LIN {X 0,Y 107.094,Z 527.487,A -85,B 0,C 180,E1 -28422.092,E2 -28422.092} C_VEL
LIN {X 0,Y 108.586,Z 526.305,A -85,B 0,C 180,E1 -28423.07,E2 -28423.07} C_VEL
LIN {X 0,Y 109.785,Z 524.448,A -85,B 0,C 180,E1 -28426.243,E2 -28426.243} C_VEL
LIN {X 0,Y 110.569,Z 522.982,A -85,B 0,C 180,E1 -28429.008,E2 -28429.008} C_VEL
LIN {X 0,Y 111.254,Z 521.399,A -85,B 0,C 180,E1 -28432.742,E2 -28432.742} C_VEL
LIN {X 0,Y 111.93,Z 520.04,A -85,B 0,C 180,E1 -28436.401,E2 -28436.401} C_VEL
LIN {X 0,Y 112.516,Z 519.038,A -85,B 0,C 180,E1 -28440.001,E2 -28440.001} C_VEL
LIN {X 0,Y 112.419,Z 518.805,A -85,B 0,C 180,E1 -28443.585,E2 -28443.585} C_VEL
LIN {X 0,Y 112.118,Z 519.081,A -85,B 0,C 180,E1 -28447.203,E2 -28447.203} C_VEL
LIN {X 0,Y 111.817,Z 519.73,A -85,B 0,C 180,E1 -28450.869,E2 -28450.869} C_VEL
LIN {X 0,Y 111.466,Z 520.726,A -85,B 0,C 180,E1 -28454.609,E2 -28454.609} C_VEL
LIN {X 0,Y 110.518,Z 523.179,A -85,B 0,C 180,E1 -28460.473,E2 -28460.473} C_VEL
LIN {X 0,Y 109.085,Z 526.099,A -85,B 0,C 180,E1 -28465.582,E2 -28465.582} C_VEL
LIN {X 0,Y 107.757,Z 528.427,A -85,B 0,C 180,E1 -28469.143,E2 -28469.143} C_VEL
LIN {X 0,Y 106.14,Z 529.943,A -85,B 0,C 180,E1 -28470.596,E2 -28470.596} C_VEL
LIN {X 0,Y 100.627,Z 533.463,A -85,B 0,C 180,E1 -28473.059,E2 -28473.059} C_VEL
LIN {X 0,Y 92.597,Z 537.838,A -85,B 0,C 180,E1 -28477.165,E2 -28477.165} C_VEL
LIN {X 0,Y 85.11,Z 541.174,A -85,B 0,C 180,E1 -28481.997,E2 -28481.997} C_VEL
LIN {X 0,Y 76.203,Z 544.136,A -85,B 0,C 180,E1 -28489.79,E2 -28489.79} C_VEL
LIN {X 0,Y 72.407,Z 545.04,A -85,B 0,C 180,E1 -28494.382,E2 -28494.382} C_VEL
LIN {X 0,Y 69.095,Z 545.527,A -85,B 0,C 180,E1 -28499.43,E2 -28499.43} C_VEL
LIN {X 0,Y 64.573,Z 545.362,A -85,B 0,C 180,E1 -28510.942,E2 -28510.942} C_VEL
LIN {X 0,Y 62.726,Z 543.678,A -85,B 0,C 180,E1 -28523.566,E2 -28523.566} C_VEL
LIN {X 0,Y 62.673,Z 542.19,A -85,B 0,C 180,E1 -28529.999,E2 -28529.999} C_VEL
LIN {X 0,Y 62.878,Z 539.11,A -85,B 0,C 180,E1 -28539.65,E2 -28539.65} C_VEL
LIN {X 0,Y 64.442,Z 534.938,A -85,B 0,C 180,E1 -28549.096,E2 -28549.096} C_VEL
LIN {X 0,Y 68.08,Z 528.537,A -85,B 0,C 180,E1 -28559.361,E2 -28559.361} C_VEL
LIN {X 0,Y 72.709,Z 521.546,A -85,B 0,C 180,E1 -28567.164,E2 -28567.164} C_VEL
LIN {X 0,Y 76.458,Z 515.745,A -85,B 0,C 180,E1 -28571.951,E2 -28571.951} C_VEL
LIN {X 0,Y 80.603,Z 509.367,A -85,B 0,C 180,E1 -28575.998,E2 -28575.998} C_VEL
LIN {X 0,Y 82.695,Z 504.549,A -85,B 0,C 180,E1 -28578.958,E2 -28578.958} C_VEL
LIN {X 0,Y 85.692,Z 495.407,A -85,B 0,C 180,E1 -28584.098,E2 -28584.098} C_VEL
LIN {X 0,Y 87.474,Z 488.295,A -85,B 0,C 180,E1 -28587.735,E2 -28587.735} C_VEL
LIN {X 0,Y 86.8,Z 482.082,A -85,B 0,C 180,E1 -28592.382,E2 -28592.382} C_VEL
LIN {X 0,Y 85.779,Z 478.507,A -85,B 0,C 180,E1 -28595.816,E2 -28595.816} C_VEL
LIN {X 0,Y 84.988,Z 476.341,A -85,B 0,C 180,E1 -28598.152,E2 -28598.152} C_VEL
LIN {X 0,Y 83.456,Z 472.714,A -85,B 0,C 180,E1 -28602.857,E2 -28602.857} C_VEL
LIN {X 0,Y 81.455,Z 468.495,A -85,B 0,C 180,E1 -28610.062,E2 -28610.062} C_VEL
LIN {X 0,Y 80.014,Z 464.504,A -85,B 0,C 180,E1 -28619.999,E2 -28619.999} C_VEL
LIN {X 0,Y 79.435,Z 464.413,A -85,B 0,C 180,E1 -28630.191,E2 -28630.191} C_VEL
LIN {X 0,Y 79.756,Z 464.688,A -85,B 0,C 180,E1 -28634.24,E2 -28634.24} C_VEL
LIN {X 0,Y 80.144,Z 467.283,A -85,B 0,C 180,E1 -28640.534,E2 -28640.534} C_VEL
LIN {X 0,Y 81.313,Z 468.944,A -85,B 0,C 180,E1 -28645.604,E2 -28645.604} C_VEL
LIN {X 0,Y 83.366,Z 473.368,A -85,B 0,C 180,E1 -28653.224,E2 -28653.224} C_VEL
LIN {X 0,Y 85.065,Z 477.902,A -85,B 0,C 180,E1 -28658.853,E2 -28658.853} C_VEL
LIN {X 0,Y 86.341,Z 481.692,A -85,B 0,C 180,E1 -28662.899,E2 -28662.899} C_VEL
LIN {X 0,Y 87.659,Z 487.537,A -85,B 0,C 180,E1 -28668.17,E2 -28668.17} C_VEL
LIN {X 0,Y 87.904,Z 488.872,A -85,B 0,C 180,E1 -28669.284,E2 -28669.284} C_VEL
LIN {X 0,Y 86.406,Z 496.526,A -85,B 0,C 180,E1 -28673.867,E2 -28673.867} C_VEL
LIN {X 0,Y 86.132,Z 497.527,A -85,B 0,C 180,E1 -28674.455,E2 -28674.455} C_VEL
LIN {X 0,Y 81.043,Z 506.139,A -85,B 0,C 180,E1 -28678.648,E2 -28678.648} C_VEL
LIN {X 0,Y 75.891,Z 514.081,A -85,B 0,C 180,E1 -28683.905,E2 -28683.905} C_VEL
LIN {X 0,Y 70.618,Z 521.83,A -85,B 0,C 180,E1 -28691.13,E2 -28691.13} C_VEL
LIN {X 0,Y 67.264,Z 527.117,A -85,B 0,C 180,E1 -28697.94,E2 -28697.94} C_VEL
LIN {X 0,Y 64.323,Z 532.25,A -85,B 0,C 180,E1 -28706.87,E2 -28706.87} C_VEL
LIN {X 0,Y 63.116,Z 534.758,A -85,B 0,C 180,E1 -28712.542,E2 -28712.542} C_VEL
LIN {X 0,Y 61.74,Z 536.654,A -85,B 0,C 180,E1 -28717.534,E2 -28717.534} C_VEL
LIN {X 0,Y 58.637,Z 539.17,A -85,B 0,C 180,E1 -28726.171,E2 -28726.171} C_VEL
LIN {X 0,Y 56.92,Z 540.71,A -85,B 0,C 180,E1 -28733.757,E2 -28733.757} C_VEL
LIN {X 0,Y 56.998,Z 541.541,A -85,B 0,C 180,E1 -28739.685,E2 -28739.685} C_VEL
LIN {X 0,Y 57.396,Z 541.749,A -85,B 0,C 180,E1 -28741.62,E2 -28741.62} C_VEL
LIN {X 0,Y 61.763,Z 542.578,A -85,B 0,C 180,E1 -28753.058,E2 -28753.058} C_VEL
LIN {X 0,Y 66.596,Z 542.319,A -85,B 0,C 180,E1 -28760.716,E2 -28760.716} C_VEL
LIN {X 0,Y 73.961,Z 540.949,A -85,B 0,C 180,E1 -28768.783,E2 -28768.783} C_VEL
LIN {X 0,Y 81.011,Z 538.875,A -85,B 0,C 180,E1 -28774.294,E2 -28774.294} C_VEL
LIN {X 0,Y 89.976,Z 535.338,A -85,B 0,C 180,E1 -28779.605,E2 -28779.605} C_VEL
LIN {X 0,Y 99.681,Z 530.427,A -85,B 0,C 180,E1 -28783.96,E2 -28783.96} C_VEL
LIN {X 0,Y 101.944,Z 529.082,A -85,B 0,C 180,E1 -28784.828,E2 -28784.828} C_VEL
LIN {X 0,Y 103.445,Z 527.812,A -85,B 0,C 180,E1 -28786.652,E2 -28786.652} C_VEL
LIN {X 0,Y 105.01,Z 525.439,A -85,B 0,C 180,E1 -28792.308,E2 -28792.308} C_VEL
LIN {X 0,Y 105.847,Z 524.124,A -85,B 0,C 180,E1 -28796.194,E2 -28796.194} C_VEL
LIN {X 0,Y 106.629,Z 523.121,A -85,B 0,C 180,E1 -28800.001,E2 -28800.001} C_VEL
LIN {X 0,Y 106.581,Z 522.939,A -85,B 0,C 180,E1 -28803.782,E2 -28803.782} C_VEL
LIN {X 0,Y 106.239,Z 523.256,A -85,B 0,C 180,E1 -28807.603,E2 -28807.603} C_VEL
LIN {X 0,Y 105.824,Z 523.945,A -85,B 0,C 180,E1 -28811.493,E2 -28811.493} C_VEL
LIN {X 0,Y 105.245,Z 525.065,A -85,B 0,C 180,E1 -28815.493,E2 -28815.493} C_VEL
LIN {X 0,Y 104.508,Z 526.648,A -85,B 0,C 180,E1 -28819.7,E2 -28819.7} C_VEL
LIN {X 0,Y 103.068,Z 528.874,A -85,B 0,C 180,E1 -28824.151,E2 -28824.151} C_VEL
LIN {X 0,Y 102.128,Z 530.228,A -85,B 0,C 180,E1 -28826.544,E2 -28826.544} C_VEL
LIN {X 0,Y 99.854,Z 531.981,A -85,B 0,C 180,E1 -28828.384,E2 -28828.384} C_VEL
LIN {X 0,Y 91.243,Z 536.629,A -85,B 0,C 180,E1 -28832.084,E2 -28832.084} C_VEL
LIN {X 0,Y 85.474,Z 539.254,A -85,B 0,C 180,E1 -28835.14,E2 -28835.14} C_VEL
LIN {X 0,Y 75.525,Z 542.811,A -85,B 0,C 180,E1 -28841.889,E2 -28841.889} C_VEL
LIN {X 0,Y 70.907,Z 544.06,A -85,B 0,C 180,E1 -28846.067,E2 -28846.067} C_VEL
LIN {X 0,Y 66.745,Z 544.905,A -85,B 0,C 180,E1 -28850.818,E2 -28850.818} C_VEL
LIN {X 0,Y 63.064,Z 545.34,A -85,B 0,C 180,E1 -28856.136,E2 -28856.136} C_VEL
LIN {X 0,Y 57.89,Z 545.102,A -85,B 0,C 180,E1 -28868.64,E2 -28868.64} C_VEL
LIN {X 0,Y 56.391,Z 544.42,A -85,B 0,C 180,E1 -28875.565,E2 -28875.565} C_VEL
LIN {X 0,Y 55.665,Z 543.309,A -85,B 0,C 180,E1 -28882.745,E2 -28882.745} C_VEL
LIN {X 0,Y 55.583,Z 541.782,A -85,B 0,C 180,E1 -28889.999,E2 -28889.999} C_VEL
LIN {X 0,Y 55.881,Z 538.622,A -85,B 0,C 180,E1 -28900.872,E2 -28900.872} C_VEL
LIN {X 0,Y 57.741,Z 534.363,A -85,B 0,C 180,E1 -28911.415,E2 -28911.415} C_VEL
LIN {X 0,Y 61.96,Z 527.87,A -85,B 0,C 180,E1 -28922.598,E2 -28922.598} C_VEL
LIN {X 0,Y 67.145,Z 520.731,A -85,B 0,C 180,E1 -28930.855,E2 -28930.855} C_VEL
LIN {X 0,Y 70.956,Z 515.28,A -85,B 0,C 180,E1 -28935.502,E2 -28935.502} C_VEL
LIN {X 0,Y 75.699,Z 508.318,A -85,B 0,C 180,E1 -28939.988,E2 -28939.988} C_VEL
LIN {X 0,Y 79.407,Z 499.352,A -85,B 0,C 180,E1 -28945.652,E2 -28945.652} C_VEL
LIN {X 0,Y 82.078,Z 490.632,A -85,B 0,C 180,E1 -28950.613,E2 -28950.613} C_VEL
LIN {X 0,Y 81.809,Z 486.001,A -85,B 0,C 180,E1 -28954.561,E2 -28954.561} C_VEL
LIN {X 0,Y 80.936,Z 482.627,A -85,B 0,C 180,E1 -28958.342,E2 -28958.342} C_VEL
LIN {X 0,Y 79.412,Z 478.104,A -85,B 0,C 180,E1 -28964.602,E2 -28964.602} C_VEL
LIN {X 0,Y 78.34,Z 475.244,A -85,B 0,C 180,E1 -28969.663,E2 -28969.663} C_VEL
LIN {X 0,Y 77.147,Z 471.217,A -85,B 0,C 180,E1 -28979.999,E2 -28979.999} C_VEL
LIN {X 0,Y 76.601,Z 470.921,A -85,B 0,C 180,E1 -28986.923,E2 -28986.923} C_VEL
LIN {X 0,Y 76.663,Z 470.972,A -85,B 0,C 180,E1 -28990.564,E2 -28990.564} C_VEL
LIN {X 0,Y 76.81,Z 472.078,A -85,B 0,C 180,E1 -28995.931,E2 -28995.931} C_VEL
LIN {X 0,Y 78.212,Z 476.052,A -85,B 0,C 180,E1 -29006.697,E2 -29006.697} C_VEL
LIN {X 0,Y 79.333,Z 479.051,A -85,B 0,C 180,E1 -29012.108,E2 -29012.108} C_VEL
LIN {X 0,Y 80.727,Z 483.727,A -85,B 0,C 180,E1 -29018.418,E2 -29018.418} C_VEL
LIN {X 0,Y 81.75,Z 488.271,A -85,B 0,C 180,E1 -29023.451,E2 -29023.451} C_VEL
LIN {X 0,Y 82.272,Z 491.778,A -85,B 0,C 180,E1 -29026.893,E2 -29026.893} C_VEL
LIN {X 0,Y 81.682,Z 494.893,A -85,B 0,C 180,E1 -29029.002,E2 -29029.002} C_VEL
LIN {X 0,Y 80.838,Z 497.854,A -85,B 0,C 180,E1 -29030.929,E2 -29030.929} C_VEL
LIN {X 0,Y 77.415,Z 503.706,A -85,B 0,C 180,E1 -29033.838,E2 -29033.838} C_VEL
LIN {X 0,Y 71.697,Z 512.082,A -85,B 0,C 180,E1 -29039.029,E2 -29039.029} C_VEL
LIN {X 0,Y 65.689,Z 520.278,A -85,B 0,C 180,E1 -29046.348,E2 -29046.348} C_VEL
LIN {X 0,Y 61.636,Z 525.845,A -85,B 0,C 180,E1 -29053.439,E2 -29053.439} C_VEL
LIN {X 0,Y 58.006,Z 531.294,A -85,B 0,C 180,E1 -29063.042,E2 -29063.042} C_VEL
LIN {X 0,Y 55.772,Z 535.57,A -85,B 0,C 180,E1 -29073.61,E2 -29073.61} C_VEL
LIN {X 0,Y 54.979,Z 538.792,A -85,B 0,C 180,E1 -29084.814,E2 -29084.814} C_VEL
LIN {X 0,Y 55.536,Z 540.396,A -85,B 0,C 180,E1 -29092.313,E2 -29092.313} C_VEL
LIN {X 0,Y 57.396,Z 541.749,A -85,B 0,C 180,E1 -29101.62,E2 -29101.62} C_VEL
LIN {X 0,Y 58.524,Z 542.322,A -85,B 0,C 180,E1 -29107.334,E2 -29107.334} C_VEL
LIN {X 0,Y 59.903,Z 542.721,A -85,B 0,C 180,E1 -29116.841,E2 -29116.841} C_VEL
LIN {X 0,Y 61.971,Z 542.598,A -85,B 0,C 180,E1 -29124.065,E2 -29124.065} C_VEL
LIN {X 0,Y 64.761,Z 542.124,A -85,B 0,C 180,E1 -29128.767,E2 -29128.767} C_VEL
LIN {X 0,Y 65.985,Z 541.881,A -85,B 0,C 180,E1 -29130.105,E2 -29130.105} C_VEL
LIN {X 0,Y 70.385,Z 541.013,A -85,B 0,C 180,E1 -29133.982,E2 -29133.982} C_VEL
LIN {X 0,Y 77.02,Z 539.182,A -85,B 0,C 180,E1 -29138.594,E2 -29138.594} C_VEL
LIN {X 0,Y 87.663,Z 535.222,A -85,B 0,C 180,E1 -29144.164,E2 -29144.164} C_VEL
LIN {X 0,Y 95.231,Z 531.591,A -85,B 0,C 180,E1 -29147.21,E2 -29147.21} C_VEL
LIN {X 0,Y 97.487,Z 530.282,A -85,B 0,C 180,E1 -29148.566,E2 -29148.566} C_VEL
LIN {X 0,Y 98.993,Z 528.515,A -85,B 0,C 180,E1 -29153.679,E2 -29153.679} C_VEL
LIN {X 0,Y 100.464,Z 526.898,A -85,B 0,C 180,E1 -29160.001,E2 -29160.001} C_VEL
LIN {X 0,Y 100.506,Z 526.711,A -85,B 0,C 180,E1 -29164.01,E2 -29164.01} C_VEL
LIN {X 0,Y 99.859,Z 527.374,A -85,B 0,C 180,E1 -29169.835,E2 -29169.835} C_VEL
LIN {X 0,Y 99.523,Z 527.862,A -85,B 0,C 180,E1 -29172.232,E2 -29172.232} C_VEL
LIN {X 0,Y 98.743,Z 529.08,A -85,B 0,C 180,E1 -29176.542,E2 -29176.542} C_VEL
LIN {X 0,Y 97.502,Z 530.784,A -85,B 0,C 180,E1 -29181.126,E2 -29181.126} C_VEL
LIN {X 0,Y 96.229,Z 532.326,A -85,B 0,C 180,E1 -29184.388,E2 -29184.388} C_VEL
LIN {X 0,Y 93.645,Z 533.826,A -85,B 0,C 180,E1 -29185.765,E2 -29185.765} C_VEL
LIN {X 0,Y 84.762,Z 538.017,A -85,B 0,C 180,E1 -29189.472,E2 -29189.472} C_VEL
LIN {X 0,Y 76.319,Z 541.185,A -85,B 0,C 180,E1 -29194.026,E2 -29194.026} C_VEL
LIN {X 0,Y 65.96,Z 543.981,A -85,B 0,C 180,E1 -29201.767,E2 -29201.767} C_VEL
LIN {X 0,Y 57.29,Z 545.154,A -85,B 0,C 180,E1 -29212.165,E2 -29212.165} C_VEL
LIN {X 0,Y 51.333,Z 544.843,A -85,B 0,C 180,E1 -29225.748,E2 -29225.748} C_VEL
LIN {X 0,Y 49.53,Z 544.098,A -85,B 0,C 180,E1 -29233.512,E2 -29233.512} C_VEL
LIN {X 0,Y 48.619,Z 542.938,A -85,B 0,C 180,E1 -29241.687,E2 -29241.687} C_VEL
LIN {X 0,Y 48.482,Z 541.374,A -85,B 0,C 180,E1 -29249.998,E2 -29249.998} C_VEL
LIN {X 0,Y 48.926,Z 538.135,A -85,B 0,C 180,E1 -29262.441,E2 -29262.441} C_VEL
LIN {X 0,Y 51.144,Z 533.786,A -85,B 0,C 180,E1 -29274.344,E2 -29274.344} C_VEL
LIN {X 0,Y 55.221,Z 528.22,A -85,B 0,C 180,E1 -29284.937,E2 -29284.937} C_VEL
LIN {X 0,Y 60.844,Z 521.251,A -85,B 0,C 180,E1 -29293.869,E2 -29293.869} C_VEL
LIN {X 0,Y 65.201,Z 515.606,A -85,B 0,C 180,E1 -29298.981,E2 -29298.981} C_VEL
LIN {X 0,Y 70.071,Z 509.105,A -85,B 0,C 180,E1 -29303.355,E2 -29303.355} C_VEL
LIN {X 0,Y 73.956,Z 501.067,A -85,B 0,C 180,E1 -29308.785,E2 -29308.785} C_VEL
LIN {X 0,Y 76.376,Z 494.81,A -85,B 0,C 180,E1 -29312.606,E2 -29312.606} C_VEL
LIN {X 0,Y 76.803,Z 493.288,A -85,B 0,C 180,E1 -29313.636,E2 -29313.636} C_VEL
LIN {X 0,Y 76.811,Z 490.588,A -85,B 0,C 180,E1 -29316.197,E2 -29316.197} C_VEL
LIN {X 0,Y 76.125,Z 486.612,A -85,B 0,C 180,E1 -29321.147,E2 -29321.147} C_VEL
LIN {X 0,Y 75.203,Z 483.316,A -85,B 0,C 180,E1 -29326.488,E2 -29326.488} C_VEL
LIN {X 0,Y 74.439,Z 480.663,A -85,B 0,C 180,E1 -29331.858,E2 -29331.858} C_VEL
LIN {X 0,Y 73.885,Z 477.752,A -85,B 0,C 180,E1 -29339.999,E2 -29339.999} C_VEL
LIN {X 0,Y 73.458,Z 477.305,A -85,B 0,C 180,E1 -29346.837,E2 -29346.837} C_VEL
LIN {X 0,Y 73.458,Z 477.474,A -85,B 0,C 180,E1 -29351.03,E2 -29351.03} C_VEL
LIN {X 0,Y 73.451,Z 478.863,A -85,B 0,C 180,E1 -29356.905,E2 -29356.905} C_VEL
LIN {X 0,Y 74.316,Z 481.733,A -85,B 0,C 180,E1 -29365.391,E2 -29365.391} C_VEL
LIN {X 0,Y 75.092,Z 484.587,A -85,B 0,C 180,E1 -29370.983,E2 -29370.983} C_VEL
LIN {X 0,Y 75.961,Z 488.576,A -85,B 0,C 180,E1 -29376.968,E2 -29376.968} C_VEL
LIN {X 0,Y 76.646,Z 493.391,A -85,B 0,C 180,E1 -29382.818,E2 -29382.818} C_VEL
LIN {X 0,Y 76.778,Z 495.332,A -85,B 0,C 180,E1 -29384.89,E2 -29384.89} C_VEL
LIN {X 0,Y 75.517,Z 499.186,A -85,B 0,C 180,E1 -29387.594,E2 -29387.594} C_VEL
LIN {X 0,Y 70.512,Z 506.659,A -85,B 0,C 180,E1 -29391.471,E2 -29391.471} C_VEL
LIN {X 0,Y 64.491,Z 514.585,A -85,B 0,C 180,E1 -29396.985,E2 -29396.985} C_VEL
LIN {X 0,Y 58.211,Z 522.31,A -85,B 0,C 180,E1 -29405.005,E2 -29405.005} C_VEL
LIN {X 0,Y 53.355,Z 528.5,A -85,B 0,C 180,E1 -29414.727,E2 -29414.727} C_VEL
LIN {X 0,Y 49.977,Z 533.401,A -85,B 0,C 180,E1 -29425.884,E2 -29425.884} C_VEL
LIN {X 0,Y 48.068,Z 537.262,A -85,B 0,C 180,E1 -29438.409,E2 -29438.409} C_VEL
LIN {X 0,Y 47.938,Z 539.248,A -85,B 0,C 180,E1 -29447.052,E2 -29447.052} C_VEL
LIN {X 0,Y 48.808,Z 540.775,A -85,B 0,C 180,E1 -29455.595,E2 -29455.595} C_VEL
LIN {X 0,Y 50.607,Z 541.852,A -85,B 0,C 180,E1 -29463.746,E2 -29463.746} C_VEL
LIN {X 0,Y 53.172,Z 542.534,A -85,B 0,C 180,E1 -29471.367,E2 -29471.367} C_VEL
LIN {X 0,Y 56.578,Z 542.808,A -85,B 0,C 180,E1 -29478.187,E2 -29478.187} C_VEL
LIN {X 0,Y 61.301,Z 542.554,A -85,B 0,C 180,E1 -29485.025,E2 -29485.025} C_VEL
LIN {X 0,Y 65.985,Z 541.881,A -85,B 0,C 180,E1 -29490.105,E2 -29490.105} C_VEL
LIN {X 0,Y 69.523,Z 541.148,A -85,B 0,C 180,E1 -29494.044,E2 -29494.044} C_VEL
LIN {X 0,Y 74.717,Z 539.484,A -85,B 0,C 180,E1 -29500.63,E2 -29500.63} C_VEL
LIN {X 0,Y 79.332,Z 537.734,A -85,B 0,C 180,E1 -29505.259,E2 -29505.259} C_VEL
LIN {X 0,Y 83.533,Z 536.067,A -85,B 0,C 180,E1 -29507.938,E2 -29507.938} C_VEL
LIN {X 0,Y 85.107,Z 535.425,A -85,B 0,C 180,E1 -29508.622,E2 -29508.622} C_VEL
LIN {X 0,Y 91.66,Z 532.443,A -85,B 0,C 180,E1 -29511.18,E2 -29511.18} C_VEL
LIN {X 0,Y 93.011,Z 531.241,A -85,B 0,C 180,E1 -29515.667,E2 -29515.667} C_VEL
LIN {X 0,Y 94.089,Z 530.342,A -85,B 0,C 180,E1 -29520.001,E2 -29520.001} C_VEL
LIN {X 0,Y 94.208,Z 530.164,A -85,B 0,C 180,E1 -29524.279,E2 -29524.279} C_VEL
LIN {X 0,Y 93.739,Z 530.579,A -85,B 0,C 180,E1 -29528.625,E2 -29528.625} C_VEL
LIN {X 0,Y 92.939,Z 531.466,A -85,B 0,C 180,E1 -29533.113,E2 -29533.113} C_VEL
LIN {X 0,Y 91.804,Z 532.745,A -85,B 0,C 180,E1 -29537.832,E2 -29537.832} C_VEL
LIN {X 0,Y 90.562,Z 534.026,A -85,B 0,C 180,E1 -29541.37,E2 -29541.37} C_VEL
LIN {X 0,Y 87.655,Z 535.483,A -85,B 0,C 180,E1 -29542.774,E2 -29542.774} C_VEL
LIN {X 0,Y 76.64,Z 539.901,A -85,B 0,C 180,E1 -29547.292,E2 -29547.292} C_VEL
LIN {X 0,Y 66.883,Z 542.751,A -85,B 0,C 180,E1 -29552.793,E2 -29552.793} C_VEL
LIN {X 0,Y 61.443,Z 543.878,A -85,B 0,C 180,E1 -29556.805,E2 -29556.805} C_VEL
LIN {X 0,Y 51.855,Z 544.969,A -85,B 0,C 180,E1 -29567.338,E2 -29567.338} C_VEL
LIN {X 0,Y 44.933,Z 544.569,A -85,B 0,C 180,E1 -29582.014,E2 -29582.014} C_VEL
LIN {X 0,Y 41.609,Z 542.565,A -85,B 0,C 180,E1 -29600.274,E2 -29600.274} C_VEL
LIN {X 0,Y 41.401,Z 540.964,A -85,B 0,C 180,E1 -29609.998,E2 -29609.998} C_VEL
LIN {X 0,Y 42.004,Z 537.642,A -85,B 0,C 180,E1 -29624.533,E2 -29624.533} C_VEL
LIN {X 0,Y 44.733,Z 533.206,A -85,B 0,C 180,E1 -29638.118,E2 -29638.118} C_VEL
LIN {X 0,Y 49.54,Z 527.547,A -85,B 0,C 180,E1 -29649.669,E2 -29649.669} C_VEL
LIN {X 0,Y 55.91,Z 520.435,A -85,B 0,C 180,E1 -29658.953,E2 -29658.953} C_VEL
LIN {X 0,Y 62.145,Z 512.95,A -85,B 0,C 180,E1 -29665.405,E2 -29665.405} C_VEL
LIN {X 0,Y 64.863,Z 509.655,A -85,B 0,C 180,E1 -29667.444,E2 -29667.444} C_VEL
LIN {X 0,Y 69.069,Z 501.961,A -85,B 0,C 180,E1 -29672.912,E2 -29672.912} C_VEL
LIN {X 0,Y 70.941,Z 497.951,A -85,B 0,C 180,E1 -29675.511,E2 -29675.511} C_VEL
LIN {X 0,Y 71.617,Z 496.061,A -85,B 0,C 180,E1 -29676.887,E2 -29676.887} C_VEL
LIN {X 0,Y 71.689,Z 493.459,A -85,B 0,C 180,E1 -29679.932,E2 -29679.932} C_VEL
LIN {X 0,Y 71.446,Z 491.498,A -85,B 0,C 180,E1 -29682.835,E2 -29682.835} C_VEL
LIN {X 0,Y 70.603,Z 487.072,A -85,B 0,C 180,E1 -29691.412,E2 -29691.412} C_VEL
LIN {X 0,Y 70.233,Z 484.057,A -85,B 0,C 180,E1 -29699.999,E2 -29699.999} C_VEL
LIN {X 0,Y 69.929,Z 483.497,A -85,B 0,C 180,E1 -29706.672,E2 -29706.672} C_VEL
LIN {X 0,Y 69.828,Z 483.842,A -85,B 0,C 180,E1 -29711.612,E2 -29711.612} C_VEL
LIN {X 0,Y 69.746,Z 485.285,A -85,B 0,C 180,E1 -29717.594,E2 -29717.594} C_VEL
LIN {X 0,Y 70.124,Z 487.154,A -85,B 0,C 180,E1 -29723.633,E2 -29723.633} C_VEL
LIN {X 0,Y 70.649,Z 489.95,A -85,B 0,C 180,E1 -29729.826,E2 -29729.826} C_VEL
LIN {X 0,Y 71.119,Z 493.953,A -85,B 0,C 180,E1 -29736.364,E2 -29736.364} C_VEL
LIN {X 0,Y 71.263,Z 497.817,A -85,B 0,C 180,E1 -29741.49,E2 -29741.49} C_VEL
LIN {X 0,Y 71.056,Z 498.998,A -85,B 0,C 180,E1 -29742.655,E2 -29742.655} C_VEL
LIN {X 0,Y 70.34,Z 500.606,A -85,B 0,C 180,E1 -29743.851,E2 -29743.851} C_VEL
LIN {X 0,Y 63.777,Z 509.394,A -85,B 0,C 180,E1 -29748.613,E2 -29748.613} C_VEL
LIN {X 0,Y 56.276,Z 518.237,A -85,B 0,C 180,E1 -29755.81,E2 -29755.81} C_VEL
LIN {X 0,Y 49.882,Z 525.287,A -85,B 0,C 180,E1 -29764.999,E2 -29764.999} C_VEL
LIN {X 0,Y 45.01,Z 530.924,A -85,B 0,C 180,E1 -29776.457,E2 -29776.457} C_VEL
LIN {X 0,Y 41.91,Z 535.374,A -85,B 0,C 180,E1 -29790.002,E2 -29790.002} C_VEL
LIN {X 0,Y 40.855,Z 537.753,A -85,B 0,C 180,E1 -29799.907,E2 -29799.907} C_VEL
LIN {X 0,Y 40.985,Z 539.686,A -85,B 0,C 180,E1 -29810.058,E2 -29810.058} C_VEL
LIN {X 0,Y 44.03,Z 541.978,A -85,B 0,C 180,E1 -29827.054,E2 -29827.054} C_VEL
LIN {X 0,Y 47.848,Z 542.811,A -85,B 0,C 180,E1 -29837.259,E2 -29837.259} C_VEL
LIN {X 0,Y 51.919,Z 543.01,A -85,B 0,C 180,E1 -29844.311,E2 -29844.311} C_VEL
LIN {X 0,Y 60.931,Z 542.237,A -85,B 0,C 180,E1 -29854.606,E2 -29854.606} C_VEL
LIN {X 0,Y 67.459,Z 541.07,A -85,B 0,C 180,E1 -29859.658,E2 -29859.658} C_VEL
LIN {X 0,Y 73.527,Z 539.485,A -85,B 0,C 180,E1 -29863.337,E2 -29863.337} C_VEL
LIN {X 0,Y 85.107,Z 535.425,A -85,B 0,C 180,E1 -29868.622,E2 -29868.622} C_VEL
LIN {X 0,Y 86.903,Z 534.626,A -85,B 0,C 180,E1 -29869.914,E2 -29869.914} C_VEL
LIN {X 0,Y 88.001,Z 533.961,A -85,B 0,C 180,E1 -29872.06,E2 -29872.06} C_VEL
LIN {X 0,Y 88.259,Z 533.581,A -85,B 0,C 180,E1 -29874.631,E2 -29874.631} C_VEL
LIN {X 0,Y 87.559,Z 533.349,A -85,B 0,C 180,E1 -29882.623,E2 -29882.623} C_VEL
LIN {X 0,Y 87.712,Z 533.282,A -85,B 0,C 180,E1 -29884.597,E2 -29884.597} C_VEL
LIN {X 0,Y 87.14,Z 533.75,A -85,B 0,C 180,E1 -29889.283,E2 -29889.283} C_VEL
LIN {X 0,Y 85.991,Z 534.699,A -85,B 0,C 180,E1 -29894.194,E2 -29894.194} C_VEL
LIN {X 0,Y 85.466,Z 535.199,A -85,B 0,C 180,E1 -29896.392,E2 -29896.392} C_VEL
LIN {X 0,Y 84.081,Z 536.097,A -85,B 0,C 180,E1 -29898.684,E2 -29898.684} C_VEL
LIN {X 0,Y 72.696,Z 540.236,A -85,B 0,C 180,E1 -29902.751,E2 -29902.751} C_VEL
LIN {X 0,Y 63.319,Z 542.701,A -85,B 0,C 180,E1 -29907.384,E2 -29907.384} C_VEL
LIN {X 0,Y 51.979,Z 544.463,A -85,B 0,C 180,E1 -29915.781,E2 -29915.781} C_VEL
LIN {X 0,Y 42.404,Z 544.731,A -85,B 0,C 180,E1 -29928.472,E2 -29928.472} C_VEL
LIN {X 0,Y 36.134,Z 543.421,A -85,B 0,C 180,E1 -29947.106,E2 -29947.106} C_VEL
LIN {X 0,Y 34.646,Z 542.186,A -85,B 0,C 180,E1 -29958.294,E2 -29958.294} C_VEL
LIN {X 0,Y 34.301,Z 540.545,A -85,B 0,C 180,E1 -29969.998,E2 -29969.998} C_VEL
LIN {X 0,Y 35.143,Z 537.136,A -85,B 0,C 180,E1 -29987.453,E2 -29987.453} C_VEL
LIN {X 0,Y 38.586,Z 532.61,A -85,B 0,C 180,E1 -30003.119,E2 -30003.119} C_VEL
LIN {X 0,Y 45.435,Z 525.72,A -85,B 0,C 180,E1 -30017.282,E2 -30017.282} C_VEL
LIN {X 0,Y 52.837,Z 518.207,A -85,B 0,C 180,E1 -30026.232,E2 -30026.232} C_VEL
LIN {X 0,Y 59.132,Z 511.159,A -85,B 0,C 180,E1 -30031.612,E2 -30031.612} C_VEL
LIN {X 0,Y 61.432,Z 507.974,A -85,B 0,C 180,E1 -30033.908,E2 -30033.908} C_VEL
LIN {X 0,Y 65.473,Z 501.253,A -85,B 0,C 180,E1 -30038.704,E2 -30038.704} C_VEL
LIN {X 0,Y 66.323,Z 499.569,A -85,B 0,C 180,E1 -30039.865,E2 -30039.865} C_VEL
LIN {X 0,Y 66.646,Z 498.071,A -85,B 0,C 180,E1 -30041.629,E2 -30041.629} C_VEL
LIN {X 0,Y 66.627,Z 496.392,A -85,B 0,C 180,E1 -30044.395,E2 -30044.395} C_VEL
LIN {X 0,Y 66.332,Z 493.263,A -85,B 0,C 180,E1 -30050.854,E2 -30050.854} C_VEL
LIN {X 0,Y 66.265,Z 492.066,A -85,B 0,C 180,E1 -30053.911,E2 -30053.911} C_VEL
LIN {X 0,Y 66.241,Z 490.146,A -85,B 0,C 180,E1 -30059.999,E2 -30059.999} C_VEL
LIN {X 0,Y 66.085,Z 489.47,A -85,B 0,C 180,E1 -30066.387,E2 -30066.387} C_VEL
LIN {X 0,Y 65.821,Z 490.06,A -85,B 0,C 180,E1 -30072.329,E2 -30072.329} C_VEL
LIN {X 0,Y 65.762,Z 492.485,A -85,B 0,C 180,E1 -30081.964,E2 -30081.964} C_VEL
LIN {X 0,Y 65.976,Z 495.246,A -85,B 0,C 180,E1 -30088.769,E2 -30088.769} C_VEL
LIN {X 0,Y 66.024,Z 498.25,A -85,B 0,C 180,E1 -30094.329,E2 -30094.329} C_VEL
LIN {X 0,Y 65.897,Z 500.836,A -85,B 0,C 180,E1 -30098.287,E2 -30098.287} C_VEL
LIN {X 0,Y 65.411,Z 502.093,A -85,B 0,C 180,E1 -30099.519,E2 -30099.519} C_VEL
LIN {X 0,Y 58.628,Z 510.425,A -85,B 0,C 180,E1 -30104.011,E2 -30104.011} C_VEL
LIN {X 0,Y 51.814,Z 517.767,A -85,B 0,C 180,E1 -30109.891,E2 -30109.891} C_VEL
LIN {X 0,Y 44.596,Z 524.981,A -85,B 0,C 180,E1 -30119.194,E2 -30119.194} C_VEL
LIN {X 0,Y 39.7,Z 529.847,A -85,B 0,C 180,E1 -30129.267,E2 -30129.267} C_VEL
LIN {X 0,Y 35.216,Z 535.058,A -85,B 0,C 180,E1 -30146.208,E2 -30146.208} C_VEL
LIN {X 0,Y 33.675,Z 538.241,A -85,B 0,C 180,E1 -30162.048,E2 -30162.048} C_VEL
LIN {X 0,Y 34.186,Z 540.094,A -85,B 0,C 180,E1 -30174.28,E2 -30174.28} C_VEL
LIN {X 0,Y 37.808,Z 542.143,A -85,B 0,C 180,E1 -30191.969,E2 -30191.969} C_VEL
LIN {X 0,Y 43.167,Z 543.076,A -85,B 0,C 180,E1 -30204.494,E2 -30204.494} C_VEL
LIN {X 0,Y 52.084,Z 543.024,A -85,B 0,C 180,E1 -30216.123,E2 -30216.123} C_VEL
LIN {X 0,Y 59.125,Z 542.236,A -85,B 0,C 180,E1 -30221.978,E2 -30221.978} C_VEL
LIN {X 0,Y 70.615,Z 539.78,A -85,B 0,C 180,E1 -30228.519,E2 -30228.519} C_VEL
LIN {X 0,Y 82.052,Z 536.025,A -85,B 0,C 180,E1 -30232.986,E2 -30232.986} C_VEL
LIN {X 0,Y 84.822,Z 534.94,A -85,B 0,C 180,E1 -30233.862,E2 -30233.862} C_VEL
LIN {X 0,Y 86.194,Z 534.255,A -85,B 0,C 180,E1 -30235.324,E2 -30235.324} C_VEL
LIN {X 0,Y 87.518,Z 533.438,A -85,B 0,C 180,E1 -30240.001,E2 -30240.001} C_VEL
LIN {X 0,Y 87.559,Z 533.349,A -85,B 0,C 180,E1 -30242.623,E2 -30242.623} C_VEL
LIN {X 0,Y 87.169,Z 533.548,A -85,B 0,C 180,E1 -30245.437,E2 -30245.437} C_VEL
LIN {X 0,Y 85.94,Z 534.18,A -85,B 0,C 180,E1 -30248.165,E2 -30248.165} C_VEL
LIN {X 0,Y 84.082,Z 535.114,A -85,B 0,C 180,E1 -30250.73,E2 -30250.73} C_VEL
LIN {X 0,Y 81.151,Z 536.5,A -85,B 0,C 180,E1 -30253.361,E2 -30253.361} C_VEL
LIN {X 0,Y 77.897,Z 537.794,A -85,B 0,C 180,E1 -30255.033,E2 -30255.033} C_VEL
LIN {X 0,Y 77.284,Z 538.012,A -85,B 0,C 180,E1 -30255.223,E2 -30255.223} C_VEL
LIN {X 0,Y 66.758,Z 541.213,A -85,B 0,C 180,E1 -30258.651,E2 -30258.651} C_VEL
LIN {X 0,Y 54.129,Z 543.662,A -85,B 0,C 180,E1 -30264.651,E2 -30264.651} C_VEL
LIN {X 0,Y 42.508,Z 544.599,A -85,B 0,C 180,E1 -30274.24,E2 -30274.24} C_VEL
LIN {X 0,Y 37.365,Z 544.479,A -85,B 0,C 180,E1 -30281.202,E2 -30281.202} C_VEL
LIN {X 0,Y 29.699,Z 543.08,A -85,B 0,C 180,E1 -30301.751,E2 -30301.751} C_VEL
LIN {X 0,Y 27.732,Z 541.807,A -85,B 0,C 180,E1 -30315.317,E2 -30315.317} C_VEL
LIN {X 0,Y 27.218,Z 540.108,A -85,B 0,C 180,E1 -30329.997,E2 -30329.997} C_VEL
LIN {X 0,Y 28.43,Z 536.62,A -85,B 0,C 180,E1 -30351.762,E2 -30351.762} C_VEL
LIN {X 0,Y 32.831,Z 531.993,A -85,B 0,C 180,E1 -30369.952,E2 -30369.952} C_VEL
LIN {X 0,Y 40.929,Z 524.974,A -85,B 0,C 180,E1 -30384.644,E2 -30384.644} C_VEL
LIN {X 0,Y 49.211,Z 517.342,A -85,B 0,C 180,E1 -30393.194,E2 -30393.194} C_VEL
LIN {X 0,Y 55.305,Z 511.001,A -85,B 0,C 180,E1 -30397.589,E2 -30397.589} C_VEL
LIN {X 0,Y 59.846,Z 504.812,A -85,B 0,C 180,E1 -30402.188,E2 -30402.188} C_VEL
LIN {X 0,Y 60.985,Z 503.037,A -85,B 0,C 180,E1 -30403.438,E2 -30403.438} C_VEL
LIN {X 0,Y 61.555,Z 501.921,A -85,B 0,C 180,E1 -30404.536,E2 -30404.536} C_VEL
LIN {X 0,Y 61.64,Z 499.289,A -85,B 0,C 180,E1 -30410.151,E2 -30410.151} C_VEL
LIN {X 0,Y 61.705,Z 497.989,A -85,B 0,C 180,E1 -30413.459,E2 -30413.459} C_VEL
LIN {X 0,Y 61.909,Z 496.015,A -85,B 0,C 180,E1 -30419.999,E2 -30419.999} C_VEL
LIN {X 0,Y 61.874,Z 495.274,A -85,B 0,C 180,E1 -30426.521,E2 -30426.521} C_VEL
LIN {X 0,Y 61.484,Z 496.029,A -85,B 0,C 180,E1 -30433.214,E2 -30433.214} C_VEL
LIN {X 0,Y 61.219,Z 497.626,A -85,B 0,C 180,E1 -30440.144,E2 -30440.144} C_VEL
LIN {X 0,Y 61.08,Z 500.222,A -85,B 0,C 180,E1 -30447.402,E2 -30447.402} C_VEL
LIN {X 0,Y 60.776,Z 502.98,A -85,B 0,C 180,E1 -30453.035,E2 -30453.035} C_VEL
LIN {X 0,Y 60.021,Z 504.624,A -85,B 0,C 180,E1 -30454.955,E2 -30454.955} C_VEL
LIN {X 0,Y 52.4,Z 512.983,A -85,B 0,C 180,E1 -30459.542,E2 -30459.542} C_VEL
LIN {X 0,Y 43.799,Z 521.168,A -85,B 0,C 180,E1 -30467.007,E2 -30467.007} C_VEL
LIN {X 0,Y 37.454,Z 526.721,A -85,B 0,C 180,E1 -30475.744,E2 -30475.744} C_VEL
LIN {X 0,Y 31.248,Z 532.162,A -85,B 0,C 180,E1 -30490.286,E2 -30490.286} C_VEL
LIN {X 0,Y 27.353,Z 536.438,A -85,B 0,C 180,E1 -30510.003,E2 -30510.003} C_VEL
LIN {X 0,Y 26.572,Z 538.719,A -85,B 0,C 180,E1 -30525.339,E2 -30525.339} C_VEL
LIN {X 0,Y 27.674,Z 540.494,A -85,B 0,C 180,E1 -30540.528,E2 -30540.528} C_VEL
LIN {X 0,Y 31.956,Z 542.306,A -85,B 0,C 180,E1 -30558.72,E2 -30558.72} C_VEL
LIN {X 0,Y 39.315,Z 543.314,A -85,B 0,C 180,E1 -30573.358,E2 -30573.358} C_VEL
LIN {X 0,Y 48.458,Z 543.255,A -85,B 0,C 180,E1 -30583.14,E2 -30583.14} C_VEL
LIN {X 0,Y 57.265,Z 542.33,A -85,B 0,C 180,E1 -30589.059,E2 -30589.059} C_VEL
LIN {X 0,Y 68.28,Z 540.087,A -85,B 0,C 180,E1 -30594.093,E2 -30594.093} C_VEL
LIN {X 0,Y 77.408,Z 537.398,A -85,B 0,C 180,E1 -30597.08,E2 -30597.08} C_VEL
LIN {X 0,Y 80.27,Z 536.332,A -85,B 0,C 180,E1 -30598.593,E2 -30598.593} C_VEL
LIN {X 0,Y 80.72,Z 536.133,A -85,B 0,C 180,E1 -30600.001,E2 -30600.001} C_VEL
LIN {X 0,Y 81.025,Z 536.023,A -85,B 0,C 180,E1 -30604.977,E2 -30604.977} C_VEL
LIN {X 0,Y 80.229,Z 536.542,A -85,B 0,C 180,E1 -30610.091,E2 -30610.091} C_VEL
LIN {X 0,Y 79.434,Z 537.082,A -85,B 0,C 180,E1 -30613.286,E2 -30613.286} C_VEL
LIN {X 0,Y 78.205,Z 537.68,A -85,B 0,C 180,E1 -30614.971,E2 -30614.971} C_VEL
LIN {X 0,Y 77.284,Z 538.012,A -85,B 0,C 180,E1 -30615.223,E2 -30615.223} C_VEL
LIN {X 0,Y 71.805,Z 539.765,A -85,B 0,C 180,E1 -30616.284,E2 -30616.284} C_VEL
LIN {X 0,Y 62.158,Z 541.999,A -85,B 0,C 180,E1 -30616.92,E2 -30616.92} C_VEL
LIN {X 0,Y 52.393,Z 543.504,A -85,B 0,C 180,E1 -30617.877,E2 -30617.877} C_VEL
LIN {X 0,Y 46.799,Z 544.011,A -85,B 0,C 180,E1 -30619.967,E2 -30619.967} C_VEL
LIN {X 0,Y 38.957,Z 544.399,A -85,B 0,C 180,E1 -30625.573,E2 -30625.573} C_VEL
LIN {X 0,Y 27.909,Z 543.666,A -85,B 0,C 180,E1 -30640.931,E2 -30640.931} C_VEL
LIN {X 0,Y 20.931,Z 541.426,A -85,B 0,C 180,E1 -30670.377,E2 -30670.377} C_VEL
LIN {X 0,Y 20.112,Z 539.648,A -85,B 0,C 180,E1 -30689.996,E2 -30689.996} C_VEL
LIN {X 0,Y 21.985,Z 536.076,A -85,B 0,C 180,E1 -30718.649,E2 -30718.649} C_VEL
LIN {X 0,Y 27.741,Z 531.35,A -85,B 0,C 180,E1 -30739.46,E2 -30739.46} C_VEL
LIN {X 0,Y 37.244,Z 524.226,A -85,B 0,C 180,E1 -30753.673,E2 -30753.673} C_VEL
LIN {X 0,Y 46.301,Z 516.546,A -85,B 0,C 180,E1 -30761.092,E2 -30761.092} C_VEL
LIN {X 0,Y 52.749,Z 510.135,A -85,B 0,C 180,E1 -30764.983,E2 -30764.983} C_VEL
LIN {X 0,Y 55.978,Z 506.118,A -85,B 0,C 180,E1 -30767.925,E2 -30767.925} C_VEL
LIN {X 0,Y 56.559,Z 505.101,A -85,B 0,C 180,E1 -30769.26,E2 -30769.26} C_VEL
LIN {X 0,Y 56.943,Z 502.586,A -85,B 0,C 180,E1 -30776.461,E2 -30776.461} C_VEL
LIN {X 0,Y 57.191,Z 501.628,A -85,B 0,C 180,E1 -30779.999,E2 -30779.999} C_VEL
LIN {X 0,Y 57.279,Z 500.875,A -85,B 0,C 180,E1 -30787.047,E2 -30787.047} C_VEL
LIN {X 0,Y 56.685,Z 501.827,A -85,B 0,C 180,E1 -30794.356,E2 -30794.356} C_VEL
LIN {X 0,Y 56.267,Z 503.667,A -85,B 0,C 180,E1 -30802.005,E2 -30802.005} C_VEL
LIN {X 0,Y 55.784,Z 505.884,A -85,B 0,C 180,E1 -30808.132,E2 -30808.132} C_VEL
LIN {X 0,Y 54.611,Z 507.53,A -85,B 0,C 180,E1 -30809.701,E2 -30809.701} C_VEL
LIN {X 0,Y 46.557,Z 515.449,A -85,B 0,C 180,E1 -30813.88,E2 -30813.88} C_VEL
LIN {X 0,Y 37.37,Z 523.164,A -85,B 0,C 180,E1 -30821.218,E2 -30821.218} C_VEL
LIN {X 0,Y 29.189,Z 529.35,A -85,B 0,C 180,E1 -30832.995,E2 -30832.995} C_VEL
LIN {X 0,Y 22.711,Z 534.281,A -85,B 0,C 180,E1 -30851.977,E2 -30851.977} C_VEL
LIN {X 0,Y 19.513,Z 538.111,A -85,B 0,C 180,E1 -30880.379,E2 -30880.379} C_VEL
LIN {X 0,Y 21.67,Z 540.895,A -85,B 0,C 180,E1 -30910.442,E2 -30910.442} C_VEL
LIN {X 0,Y 26.781,Z 542.475,A -85,B 0,C 180,E1 -30928.345,E2 -30928.345} C_VEL
LIN {X 0,Y 36.586,Z 543.549,A -85,B 0,C 180,E1 -30943.839,E2 -30943.839} C_VEL
LIN {X 0,Y 45.643,Z 543.488,A -85,B 0,C 180,E1 -30951.144,E2 -30951.144} C_VEL
LIN {X 0,Y 56.328,Z 542.396,A -85,B 0,C 180,E1 -30956.528,E2 -30956.528} C_VEL
LIN {X 0,Y 66.704,Z 540.376,A -85,B 0,C 180,E1 -30960.001,E2 -30960.001} C_VEL
LIN {X 0,Y 70.29,Z 539.456,A -85,B 0,C 180,E1 -30960.963,E2 -30960.963} C_VEL
LIN {X 0,Y 74.107,Z 538.341,A -85,B 0,C 180,E1 -30963.176,E2 -30963.176} C_VEL
LIN {X 0,Y 74.115,Z 538.378,A -85,B 0,C 180,E1 -30965.442,E2 -30965.442} C_VEL
LIN {X 0,Y 73.517,Z 538.719,A -85,B 0,C 180,E1 -30969.335,E2 -30969.335} C_VEL
LIN {X 0,Y 71.576,Z 539.398,A -85,B 0,C 180,E1 -30970.919,E2 -30970.919} C_VEL
LIN {X 0,Y 64.834,Z 541.191,A -85,B 0,C 180,E1 -30972.683,E2 -30972.683} C_VEL
LIN {X 0,Y 51.57,Z 543.554,A -85,B 0,C 180,E1 -30977.451,E2 -30977.451} C_VEL
LIN {X 0,Y 46.799,Z 544.011,A -85,B 0,C 180,E1 -30979.967,E2 -30979.967} C_VEL
LIN {X 0,Y 41.28,Z 544.35,A -85,B 0,C 180,E1 -30982.665,E2 -30982.665} C_VEL
LIN {X 0,Y 31.643,Z 544.183,A -85,B 0,C 180,E1 -30986.322,E2 -30986.322} C_VEL
LIN {X 0,Y 24.061,Z 543.432,A -85,B 0,C 180,E1 -30991.029,E2 -30991.029} C_VEL
LIN {X 0,Y 19.01,Z 542.527,A -85,B 0,C 180,E1 -30998.937,E2 -30998.937} C_VEL
LIN {X 0,Y 17.62,Z 542.163,A -85,B 0,C 180,E1 -31003.166,E2 -31003.166} C_VEL
LIN {X 0,Y 14.443,Z 541.02,A -85,B 0,C 180,E1 -31020.877,E2 -31020.877} C_VEL
LIN {X 0,Y 13.008,Z 539.187,A -85,B 0,C 180,E1 -31049.994,E2 -31049.994} C_VEL
LIN {X 0,Y 16.09,Z 535.525,A -85,B 0,C 180,E1 -31090.927,E2 -31090.927} C_VEL
LIN {X 0,Y 23.721,Z 530.705,A -85,B 0,C 180,E1 -31112.718,E2 -31112.718} C_VEL
LIN {X 0,Y 33.056,Z 524.61,A -85,B 0,C 180,E1 -31123.076,E2 -31123.076} C_VEL
LIN {X 0,Y 42.938,Z 516.984,A -85,B 0,C 180,E1 -31129.118,E2 -31129.118} C_VEL
LIN {X 0,Y 49.66,Z 510.787,A -85,B 0,C 180,E1 -31132.139,E2 -31132.139} C_VEL
LIN {X 0,Y 50.68,Z 509.708,A -85,B 0,C 180,E1 -31132.898,E2 -31132.898} C_VEL
LIN {X 0,Y 51.645,Z 508.503,A -85,B 0,C 180,E1 -31134.282,E2 -31134.282} C_VEL
LIN {X 0,Y 52.158,Z 506.961,A -85,B 0,C 180,E1 -31139.999,E2 -31139.999} C_VEL
LIN {X 0,Y 52.341,Z 506.202,A -85,B 0,C 180,E1 -31147.715,E2 -31147.715} C_VEL
LIN {X 0,Y 51.389,Z 507.669,A -85,B 0,C 180,E1 -31156.809,E2 -31156.809} C_VEL
LIN {X 0,Y 51.222,Z 508.319,A -85,B 0,C 180,E1 -31160.049,E2 -31160.049} C_VEL
LIN {X 0,Y 49.761,Z 510.248,A -85,B 0,C 180,E1 -31163.366,E2 -31163.366} C_VEL
LIN {X 0,Y 39.668,Z 519.087,A -85,B 0,C 180,E1 -31167.651,E2 -31167.651} C_VEL
LIN {X 0,Y 29.95,Z 526.127,A -85,B 0,C 180,E1 -31174.792,E2 -31174.792} C_VEL
LIN {X 0,Y 20.992,Z 531.764,A -85,B 0,C 180,E1 -31187.97,E2 -31187.97} C_VEL
LIN {X 0,Y 15.065,Z 535.515,A -85,B 0,C 180,E1 -31208.899,E2 -31208.899} C_VEL
LIN {X 0,Y 13.048,Z 539.609,A -85,B 0,C 180,E1 -31262.596,E2 -31262.596} C_VEL
LIN {X 0,Y 16.774,Z 541.297,A -85,B 0,C 180,E1 -31286.931,E2 -31286.931} C_VEL
LIN {X 0,Y 22.639,Z 542.635,A -85,B 0,C 180,E1 -31301.917,E2 -31301.917} C_VEL
LIN {X 0,Y 35.248,Z 543.784,A -85,B 0,C 180,E1 -31315.516,E2 -31315.516} C_VEL
LIN {X 0,Y 43.79,Z 543.724,A -85,B 0,C 180,E1 -31320.002,E2 -31320.002} C_VEL
LIN {X 0,Y 56.369,Z 542.46,A -85,B 0,C 180,E1 -31324.115,E2 -31324.115} C_VEL
LIN {X 0,Y 63.567,Z 541.158,A -85,B 0,C 180,E1 -31325.705,E2 -31325.705} C_VEL
LIN {X 0,Y 64.426,Z 540.996,A -85,B 0,C 180,E1 -31326.264,E2 -31326.264} C_VEL
LIN {X 0,Y 56.759,Z 542.495,A -85,B 0,C 180,E1 -31327.87,E2 -31327.87} C_VEL
LIN {X 0,Y 43.124,Z 544.019,A -85,B 0,C 180,E1 -31332.083,E2 -31332.083} C_VEL
LIN {X 0,Y 29.961,Z 543.953,A -85,B 0,C 180,E1 -31340.228,E2 -31340.228} C_VEL
LIN {X 0,Y 18.442,Z 542.4,A -85,B 0,C 180,E1 -31360.338,E2 -31360.338} C_VEL
LIN {X 0,Y 17.62,Z 542.163,A -85,B 0,C 180,E1 -31363.166,E2 -31363.166} C_VEL
LIN {X 0,Y 13.768,Z 540.989,A -85,B 0,C 180,E1 -31378.946,E2 -31378.946} C_VEL
LIN {X 0,Y 10.465,Z 539.471,A -85,B 0,C 180,E1 -31401.59,E2 -31401.59} C_VEL
LIN {X 0,Y 11.079,Z 535.615,A -85,B 0,C 180,E1 -31465.882,E2 -31465.882} C_VEL
LIN {X 0,Y 15.257,Z 533.273,A -85,B 0,C 180,E1 -31482.285,E2 -31482.285} C_VEL
LIN {X 0,Y 16.914,Z 532.422,A -85,B 0,C 180,E1 -31485.145,E2 -31485.145} C_VEL
LIN {X 0,Y 28.258,Z 526.109,A -85,B 0,C 180,E1 -31494.136,E2 -31494.136} C_VEL
LIN {X 0,Y 38.678,Z 518.862,A -85,B 0,C 180,E1 -31497.874,E2 -31497.874} C_VEL
LIN {X 0,Y 46.782,Z 512.055,A -85,B 0,C 180,E1 -31499.998,E2 -31499.998} C_VEL
LIN {X 0,Y 46.944,Z 511.414,A -85,B 0,C 180,E1 -31508.609,E2 -31508.609} C_VEL
LIN {X 0,Y 46.539,Z 511.846,A -85,B 0,C 180,E1 -31511.884,E2 -31511.884} C_VEL
LIN {X 0,Y 45.01,Z 513.409,A -85,B 0,C 180,E1 -31515.88,E2 -31515.88} C_VEL
LIN {X 0,Y 35.166,Z 521.18,A -85,B 0,C 180,E1 -31518.334,E2 -31518.334} C_VEL
LIN {X 0,Y 24.831,Z 527.862,A -85,B 0,C 180,E1 -31523.104,E2 -31523.104} C_VEL
LIN {X 0,Y 13.132,Z 533.973,A -85,B 0,C 180,E1 -31536.613,E2 -31536.613} C_VEL
LIN {X 0,Y 5.451,Z 537.982,A -85,B 0,C 180,E1 -31590.014,E2 -31590.014} C_VEL
LIN {X 0,Y 7.923,Z 540.054,A -85,B 0,C 180,E1 -31652.529,E2 -31652.529} C_VEL
LIN {X 0,Y 14.168,Z 541.7,A -85,B 0,C 180,E1 -31672.812,E2 -31672.812} C_VEL
LIN {X 0,Y 21.086,Z 542.903,A -85,B 0,C 180,E1 -31680.699,E2 -31680.699} C_VEL
LIN {X 0,Y 28.22,Z 543.662,A -85,B 0,C 180,E1 -31684.986,E2 -31684.986} C_VEL
LIN {X 0,Y 28.298,Z 543.691,A -85,B 0,C 180,E1 -31686.566,E2 -31686.566} C_VEL
LIN {X 0,Y 14.866,Z 542.051,A -85,B 0,C 180,E1 -31698.989,E2 -31698.989} C_VEL
LIN {X 0,Y 8.943,Z 540.601,A -85,B 0,C 180,E1 -31718.186,E2 -31718.186} C_VEL
LIN {X 0,Y 5.914,Z 538.726,A -85,B 0,C 180,E1 -31769.987,E2 -31769.987} C_VEL
LIN {X 0,Y 11.68,Z 534.977,A -85,B 0,C 180,E1 -31834.476,E2 -31834.476} C_VEL
LIN {X 0,Y 16.914,Z 532.422,A -85,B 0,C 180,E1 -31845.145,E2 -31845.145} C_VEL
LIN {X 0,Y 19.568,Z 534.239,A -85,B 0,C 180,E1 -31848.291,E2 -31848.291} C_VEL
LIN {X 0,Y 19.568,Z 600,A -85,B 0,C 180,E1 -31848.291,E2 -31848.291} C_VEL
LIN {X 0,Y 19.568,Z 600,A -85,B 0,C 180,E1 -31848.291,E2 -31848.291}

QRS_NEXT_CUT()

QRS_NEXT()
QRS_HOME()

END
